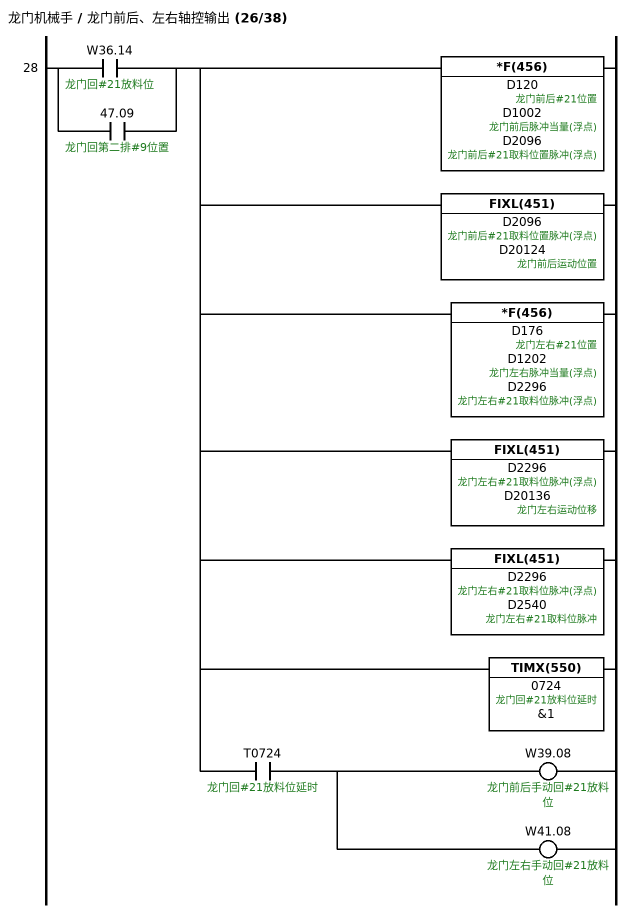
; [picture p353: 龙门机械手 / 龙门前后、左右轴控输出, rungs 28-28]
; rung 28
LD W36.14  ; 龙门回#21放料位
OR 47.09  ; 龙门回第二排#9位置
*F(456) D120 D1002 D2096  ; 龙门前后#21位置, 龙门前后脉冲当量(浮点), 龙门前后#21取料位置脉冲(浮点)
FIXL(451) D2096 D20124  ; 龙门前后#21取料位置脉冲(浮点), 龙门前后运动位置
*F(456) D176 D1202 D2296  ; 龙门左右#21位置, 龙门左右脉冲当量(浮点), 龙门左右#21取料位脉冲(浮点)
FIXL(451) D2296 D20136  ; 龙门左右#21取料位脉冲(浮点), 龙门左右运动位移
FIXL(451) D2296 D2540  ; 龙门左右#21取料位脉冲(浮点), 龙门左右#21取料位脉冲
TIMX(550) 0724 &1  ; 龙门回#21放料位延时
AND T0724  ; 龙门回#21放料位延时
OUT W39.08  ; 龙门前后手动回#21放料位
OUT W41.08  ; 龙门左右手动回#21放料位

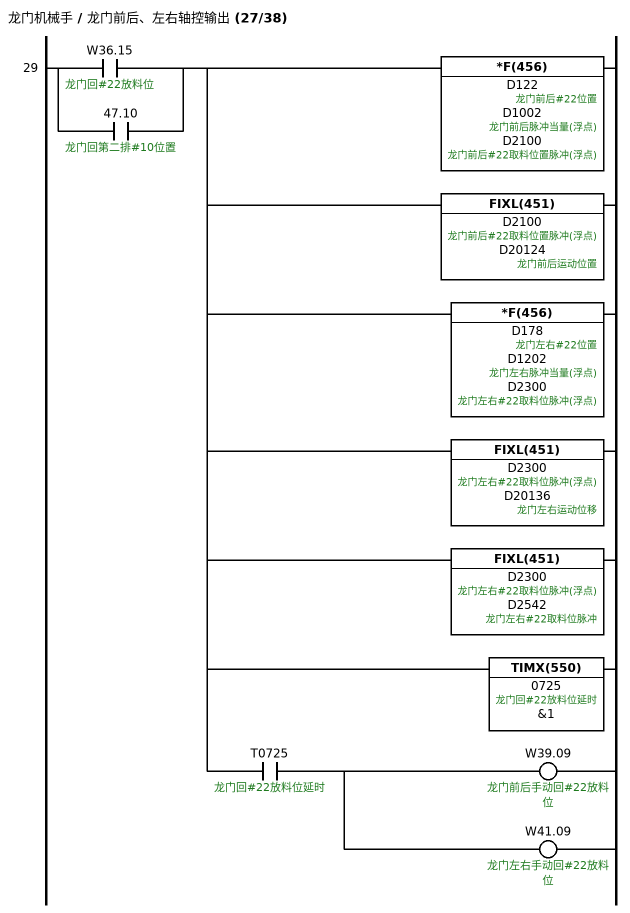
; rung 29
LD W36.15  ; 龙门回#22放料位
OR 47.10  ; 龙门回第二排#10位置
*F(456) D122 D1002 D2100  ; 龙门前后#22位置, 龙门前后脉冲当量(浮点), 龙门前后#22取料位置脉冲(浮点)
FIXL(451) D2100 D20124  ; 龙门前后#22取料位置脉冲(浮点), 龙门前后运动位置
*F(456) D178 D1202 D2300  ; 龙门左右#22位置, 龙门左右脉冲当量(浮点), 龙门左右#22取料位脉冲(浮点)
FIXL(451) D2300 D20136  ; 龙门左右#22取料位脉冲(浮点), 龙门左右运动位移
FIXL(451) D2300 D2542  ; 龙门左右#22取料位脉冲(浮点), 龙门左右#22取料位脉冲
TIMX(550) 0725 &1  ; 龙门回#22放料位延时
AND T0725  ; 龙门回#22放料位延时
OUT W39.09  ; 龙门前后手动回#22放料位
OUT W41.09  ; 龙门左右手动回#22放料位

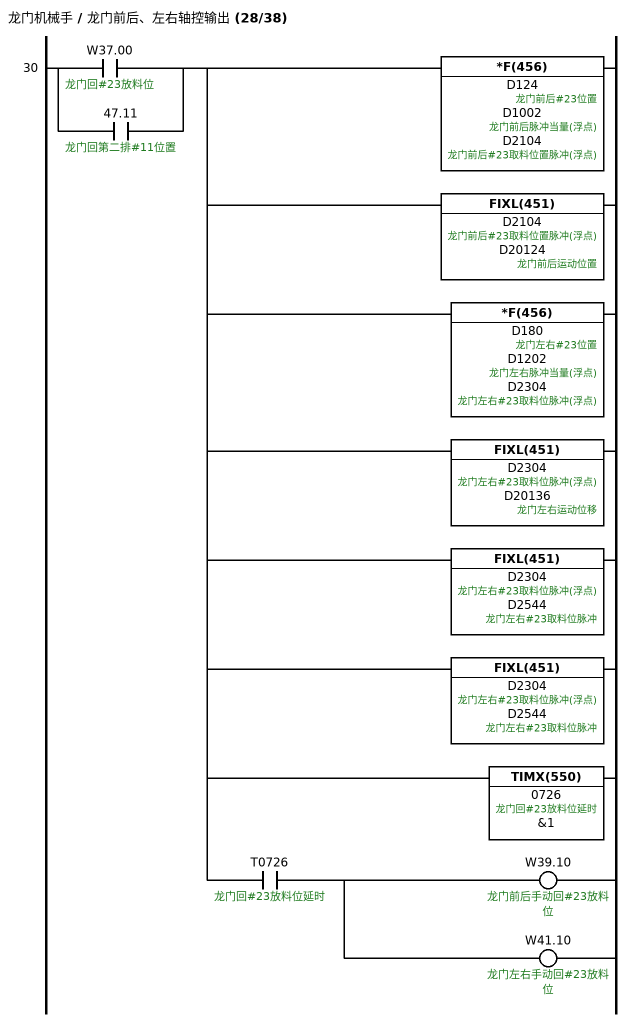
; rung 30
LD W37.00  ; 龙门回#23放料位
OR 47.11  ; 龙门回第二排#11位置
*F(456) D124 D1002 D2104  ; 龙门前后#23位置, 龙门前后脉冲当量(浮点), 龙门前后#23取料位置脉冲(浮点)
FIXL(451) D2104 D20124  ; 龙门前后#23取料位置脉冲(浮点), 龙门前后运动位置
*F(456) D180 D1202 D2304  ; 龙门左右#23位置, 龙门左右脉冲当量(浮点), 龙门左右#23取料位脉冲(浮点)
FIXL(451) D2304 D20136  ; 龙门左右#23取料位脉冲(浮点), 龙门左右运动位移
FIXL(451) D2304 D2544  ; 龙门左右#23取料位脉冲(浮点), 龙门左右#23取料位脉冲
FIXL(451) D2304 D2544  ; 龙门左右#23取料位脉冲(浮点), 龙门左右#23取料位脉冲
TIMX(550) 0726 &1  ; 龙门回#23放料位延时
AND T0726  ; 龙门回#23放料位延时
OUT W39.10  ; 龙门前后手动回#23放料位
OUT W41.10  ; 龙门左右手动回#23放料位

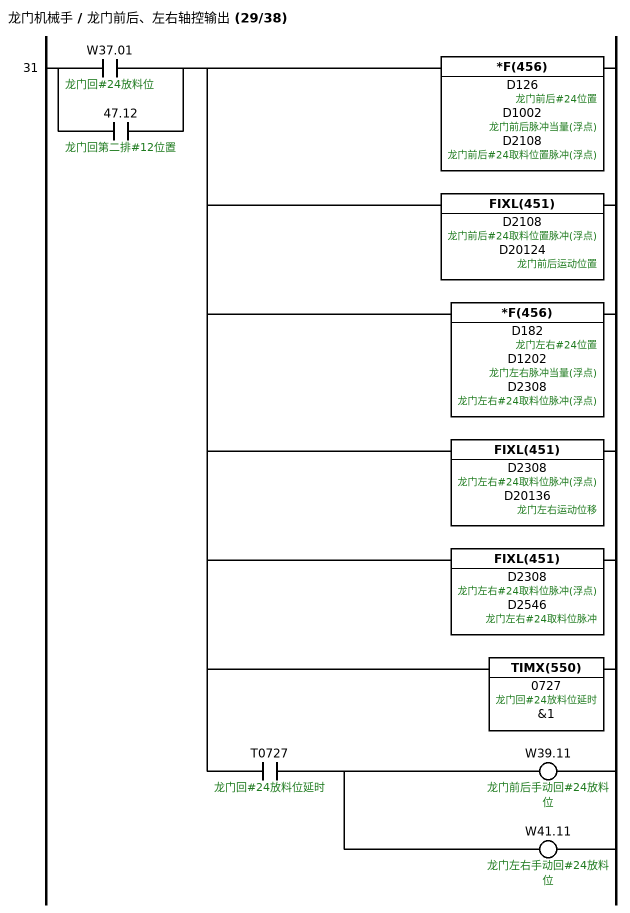
; rung 31
LD W37.01  ; 龙门回#24放料位
OR 47.12  ; 龙门回第二排#12位置
*F(456) D126 D1002 D2108  ; 龙门前后#24位置, 龙门前后脉冲当量(浮点), 龙门前后#24取料位置脉冲(浮点)
FIXL(451) D2108 D20124  ; 龙门前后#24取料位置脉冲(浮点), 龙门前后运动位置
*F(456) D182 D1202 D2308  ; 龙门左右#24位置, 龙门左右脉冲当量(浮点), 龙门左右#24取料位脉冲(浮点)
FIXL(451) D2308 D20136  ; 龙门左右#24取料位脉冲(浮点), 龙门左右运动位移
FIXL(451) D2308 D2546  ; 龙门左右#24取料位脉冲(浮点), 龙门左右#24取料位脉冲
TIMX(550) 0727 &1  ; 龙门回#24放料位延时
AND T0727  ; 龙门回#24放料位延时
OUT W39.11  ; 龙门前后手动回#24放料位
OUT W41.11  ; 龙门左右手动回#24放料位

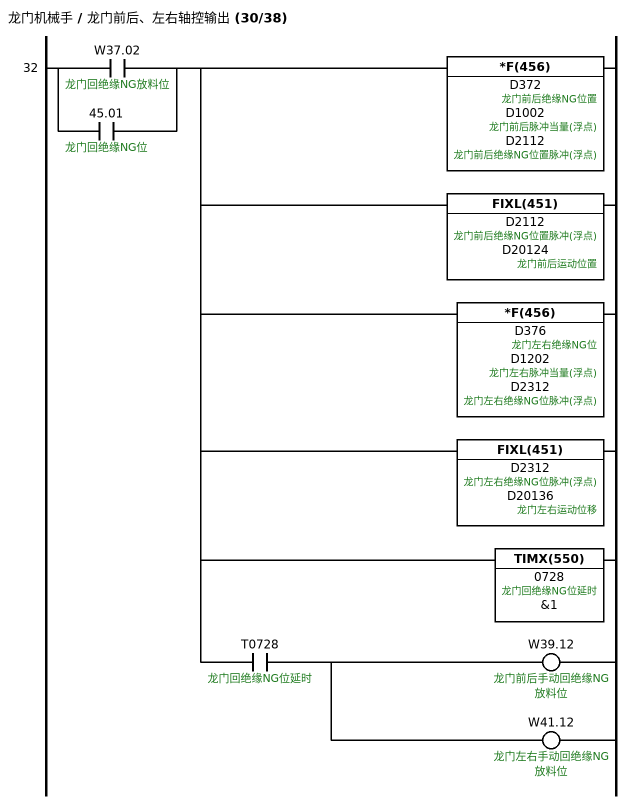
; rung 32
LD W37.02  ; 龙门回绝缘NG放料位
OR 45.01  ; 龙门回绝缘NG位
*F(456) D372 D1002 D2112  ; 龙门前后绝缘NG位置, 龙门前后脉冲当量(浮点), 龙门前后绝缘NG位置脉冲(浮点)
FIXL(451) D2112 D20124  ; 龙门前后绝缘NG位置脉冲(浮点), 龙门前后运动位置
*F(456) D376 D1202 D2312  ; 龙门左右绝缘NG位, 龙门左右脉冲当量(浮点), 龙门左右绝缘NG位脉冲(浮点)
FIXL(451) D2312 D20136  ; 龙门左右绝缘NG位脉冲(浮点), 龙门左右运动位移
TIMX(550) 0728 &1  ; 龙门回绝缘NG位延时
AND T0728  ; 龙门回绝缘NG位延时
OUT W39.12  ; 龙门前后手动回绝缘NG放料位
OUT W41.12  ; 龙门左右手动回绝缘NG放料位

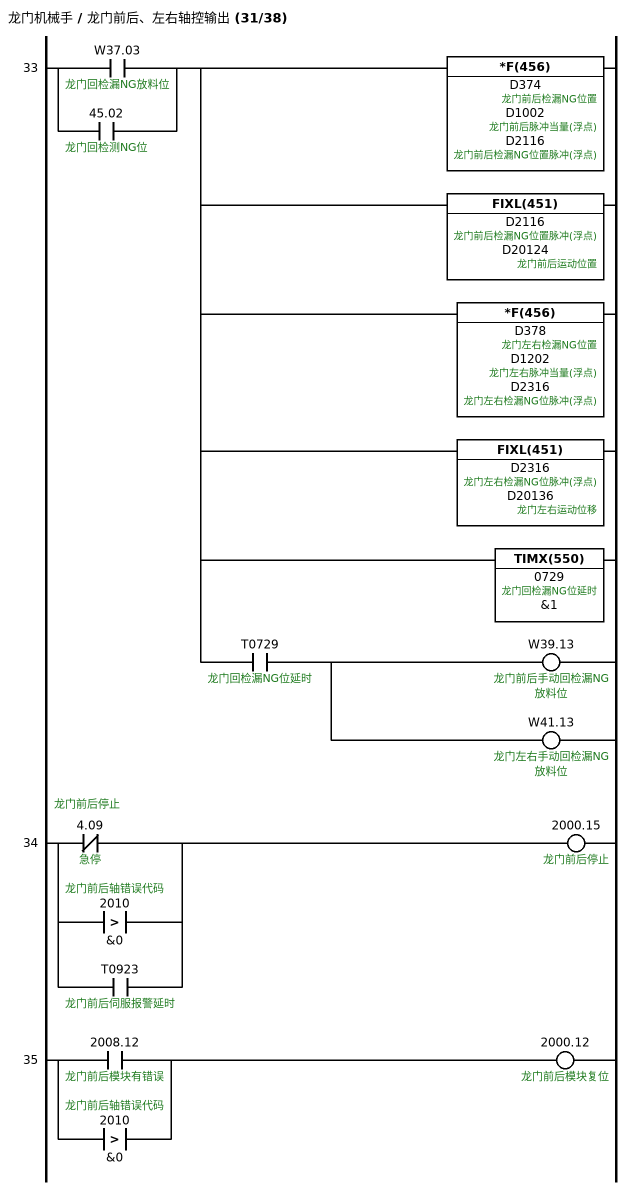
; rung 33
LD W37.03  ; 龙门回检漏NG放料位
OR 45.02  ; 龙门回检测NG位
*F(456) D374 D1002 D2116  ; 龙门前后检漏NG位置, 龙门前后脉冲当量(浮点), 龙门前后检漏NG位置脉冲(浮点)
FIXL(451) D2116 D20124  ; 龙门前后检漏NG位置脉冲(浮点), 龙门前后运动位置
*F(456) D378 D1202 D2316  ; 龙门左右检漏NG位置, 龙门左右脉冲当量(浮点), 龙门左右检漏NG位脉冲(浮点)
FIXL(451) D2316 D20136  ; 龙门左右检漏NG位脉冲(浮点), 龙门左右运动位移
TIMX(550) 0729 &1  ; 龙门回检漏NG位延时
AND T0729  ; 龙门回检漏NG位延时
OUT W39.13  ; 龙门前后手动回检漏NG放料位
OUT W41.13  ; 龙门左右手动回检漏NG放料位
; rung 34: 龙门前后停止
LDNOT 4.09  ; 急停
OR>(320) 2010 &0  ; 龙门前后轴错误代码
OR T0923  ; 龙门前后伺服报警延时
OUT 2000.15  ; 龙门前后停止
; rung 35
LD 2008.12  ; 龙门前后模块有错误
OR>(320) 2010 &0  ; 龙门前后轴错误代码
OUT 2000.12  ; 龙门前后模块复位

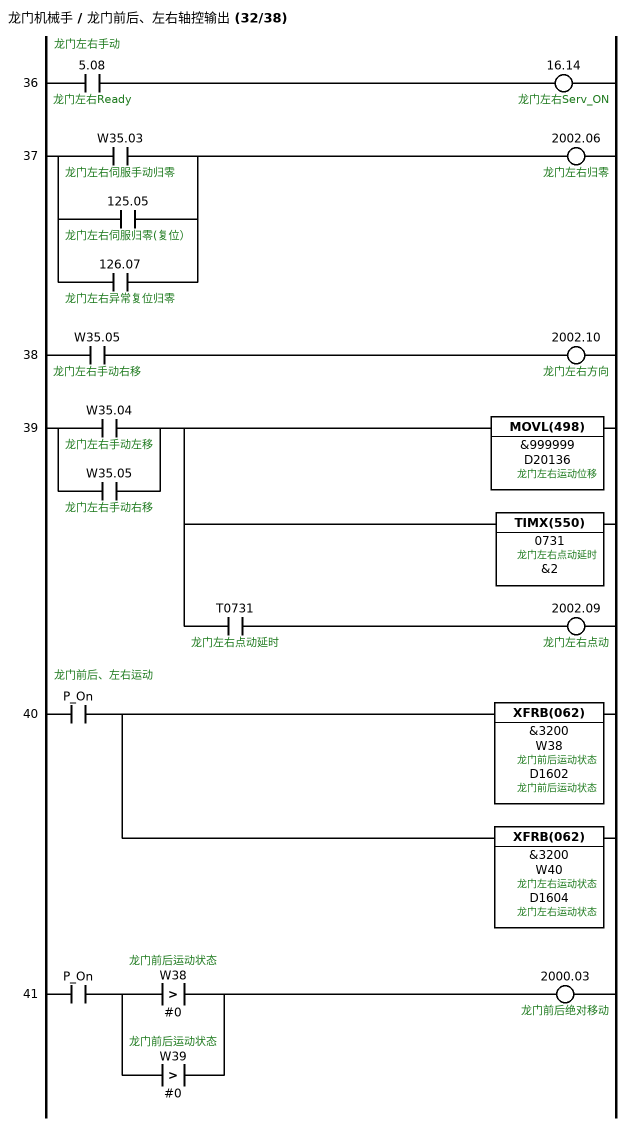
; rung 36: 龙门左右手动
LD 5.08  ; 龙门左右Ready
OUT 16.14  ; 龙门左右Serv_ON
; rung 37
LD W35.03  ; 龙门左右伺服手动归零
OR 125.05  ; 龙门左右伺服归零(复位）
OR 126.07  ; 龙门左右异常复位归零
OUT 2002.06  ; 龙门左右归零
; rung 38
LD W35.05  ; 龙门左右手动右移
OUT 2002.10  ; 龙门左右方向
; rung 39
LD W35.04  ; 龙门左右手动左移
OR W35.05  ; 龙门左右手动右移
MOVL(498) &999999 D20136  ; 龙门左右运动位移
TIMX(550) 0731 &2  ; 龙门左右点动延时
AND T0731  ; 龙门左右点动延时
OUT 2002.09  ; 龙门左右点动
; rung 40: 龙门前后、左右运动
LD P_On
XFRB(062) &3200 W38 D1602  ; 龙门前后运动状态
XFRB(062) &3200 W40 D1604  ; 龙门左右运动状态
; rung 41
LD P_On
LD>(320) W38 #0  ; 龙门前后运动状态
OR>(320) W39 #0  ; 龙门前后运动状态
ANDLD
OUT 2000.03  ; 龙门前后绝对移动

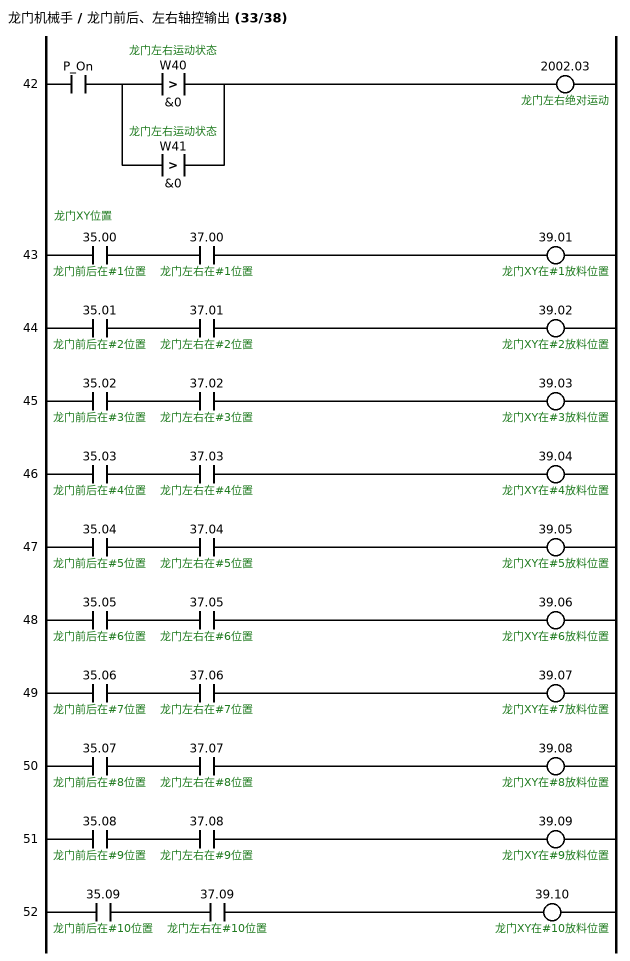
; rung 42
LD P_On
LD>(320) W40 &0  ; 龙门左右运动状态
OR>(320) W41 &0  ; 龙门左右运动状态
ANDLD
OUT 2002.03  ; 龙门左右绝对运动
; rung 43: 龙门XY位置
LD 35.00  ; 龙门前后在#1位置
AND 37.00  ; 龙门左右在#1位置
OUT 39.01  ; 龙门XY在#1放料位置
; rung 44
LD 35.01  ; 龙门前后在#2位置
AND 37.01  ; 龙门左右在#2位置
OUT 39.02  ; 龙门XY在#2放料位置
; rung 45
LD 35.02  ; 龙门前后在#3位置
AND 37.02  ; 龙门左右在#3位置
OUT 39.03  ; 龙门XY在#3放料位置
; rung 46
LD 35.03  ; 龙门前后在#4位置
AND 37.03  ; 龙门左右在#4位置
OUT 39.04  ; 龙门XY在#4放料位置
; rung 47
LD 35.04  ; 龙门前后在#5位置
AND 37.04  ; 龙门左右在#5位置
OUT 39.05  ; 龙门XY在#5放料位置
; rung 48
LD 35.05  ; 龙门前后在#6位置
AND 37.05  ; 龙门左右在#6位置
OUT 39.06  ; 龙门XY在#6放料位置
; rung 49
LD 35.06  ; 龙门前后在#7位置
AND 37.06  ; 龙门左右在#7位置
OUT 39.07  ; 龙门XY在#7放料位置
; rung 50
LD 35.07  ; 龙门前后在#8位置
AND 37.07  ; 龙门左右在#8位置
OUT 39.08  ; 龙门XY在#8放料位置
; rung 51
LD 35.08  ; 龙门前后在#9位置
AND 37.08  ; 龙门左右在#9位置
OUT 39.09  ; 龙门XY在#9放料位置
; rung 52
LD 35.09  ; 龙门前后在#10位置
AND 37.09  ; 龙门左右在#10位置
OUT 39.10  ; 龙门XY在#10放料位置

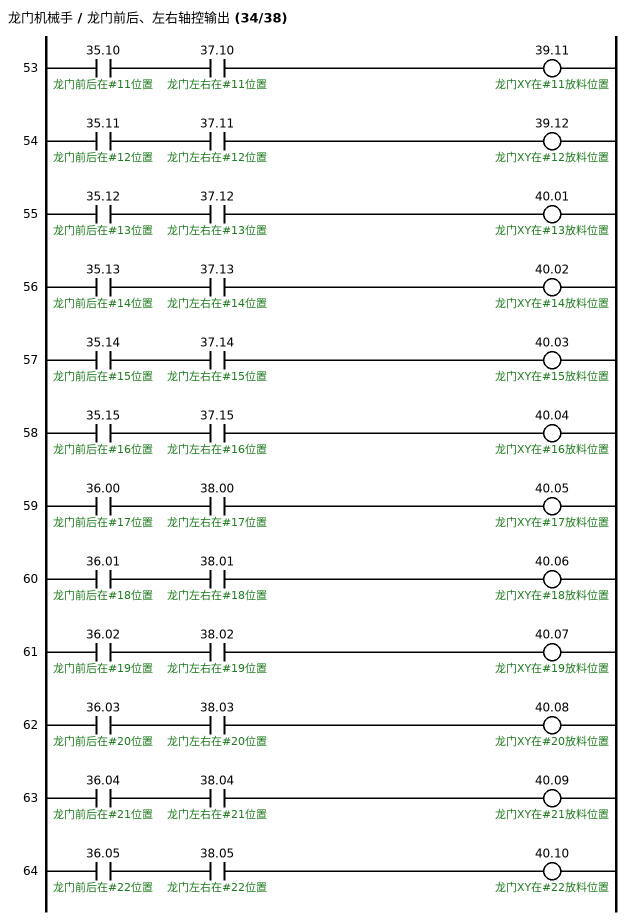
; rung 53
LD 35.10  ; 龙门前后在#11位置
AND 37.10  ; 龙门左右在#11位置
OUT 39.11  ; 龙门XY在#11放料位置
; rung 54
LD 35.11  ; 龙门前后在#12位置
AND 37.11  ; 龙门左右在#12位置
OUT 39.12  ; 龙门XY在#12放料位置
; rung 55
LD 35.12  ; 龙门前后在#13位置
AND 37.12  ; 龙门左右在#13位置
OUT 40.01  ; 龙门XY在#13放料位置
; rung 56
LD 35.13  ; 龙门前后在#14位置
AND 37.13  ; 龙门左右在#14位置
OUT 40.02  ; 龙门XY在#14放料位置
; rung 57
LD 35.14  ; 龙门前后在#15位置
AND 37.14  ; 龙门左右在#15位置
OUT 40.03  ; 龙门XY在#15放料位置
; rung 58
LD 35.15  ; 龙门前后在#16位置
AND 37.15  ; 龙门左右在#16位置
OUT 40.04  ; 龙门XY在#16放料位置
; rung 59
LD 36.00  ; 龙门前后在#17位置
AND 38.00  ; 龙门左右在#17位置
OUT 40.05  ; 龙门XY在#17放料位置
; rung 60
LD 36.01  ; 龙门前后在#18位置
AND 38.01  ; 龙门左右在#18位置
OUT 40.06  ; 龙门XY在#18放料位置
; rung 61
LD 36.02  ; 龙门前后在#19位置
AND 38.02  ; 龙门左右在#19位置
OUT 40.07  ; 龙门XY在#19放料位置
; rung 62
LD 36.03  ; 龙门前后在#20位置
AND 38.03  ; 龙门左右在#20位置
OUT 40.08  ; 龙门XY在#20放料位置
; rung 63
LD 36.04  ; 龙门前后在#21位置
AND 38.04  ; 龙门左右在#21位置
OUT 40.09  ; 龙门XY在#21放料位置
; rung 64
LD 36.05  ; 龙门前后在#22位置
AND 38.05  ; 龙门左右在#22位置
OUT 40.10  ; 龙门XY在#22放料位置

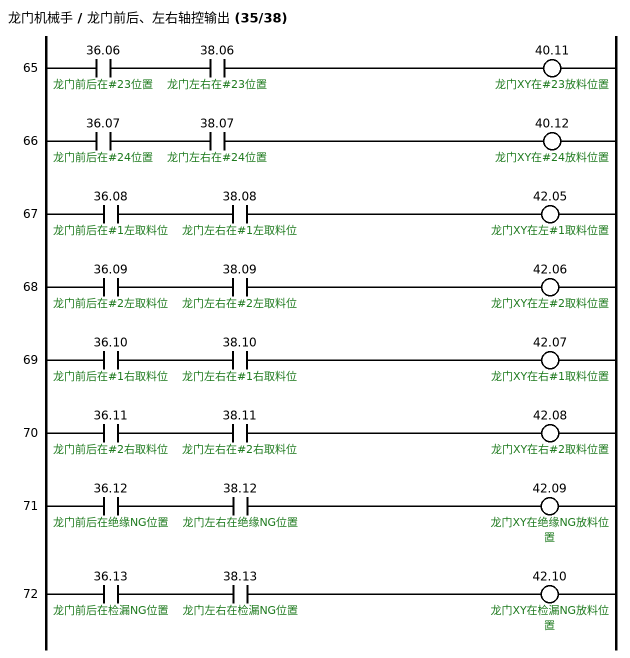
; rung 65
LD 36.06  ; 龙门前后在#23位置
AND 38.06  ; 龙门左右在#23位置
OUT 40.11  ; 龙门XY在#23放料位置
; rung 66
LD 36.07  ; 龙门前后在#24位置
AND 38.07  ; 龙门左右在#24位置
OUT 40.12  ; 龙门XY在#24放料位置
; rung 67
LD 36.08  ; 龙门前后在#1左取料位
AND 38.08  ; 龙门左右在#1左取料位
OUT 42.05  ; 龙门XY在左#1取料位置
; rung 68
LD 36.09  ; 龙门前后在#2左取料位
AND 38.09  ; 龙门左右在#2左取料位
OUT 42.06  ; 龙门XY在左#2取料位置
; rung 69
LD 36.10  ; 龙门前后在#1右取料位
AND 38.10  ; 龙门左右在#1右取料位
OUT 42.07  ; 龙门XY在右#1取料位置
; rung 70
LD 36.11  ; 龙门前后在#2右取料位
AND 38.11  ; 龙门左右在#2右取料位
OUT 42.08  ; 龙门XY在右#2取料位置
; rung 71
LD 36.12  ; 龙门前后在绝缘NG位置
AND 38.12  ; 龙门左右在绝缘NG位置
OUT 42.09  ; 龙门XY在绝缘NG放料位置
; rung 72
LD 36.13  ; 龙门前后在检漏NG位置
AND 38.13  ; 龙门左右在检漏NG位置
OUT 42.10  ; 龙门XY在检漏NG放料位置

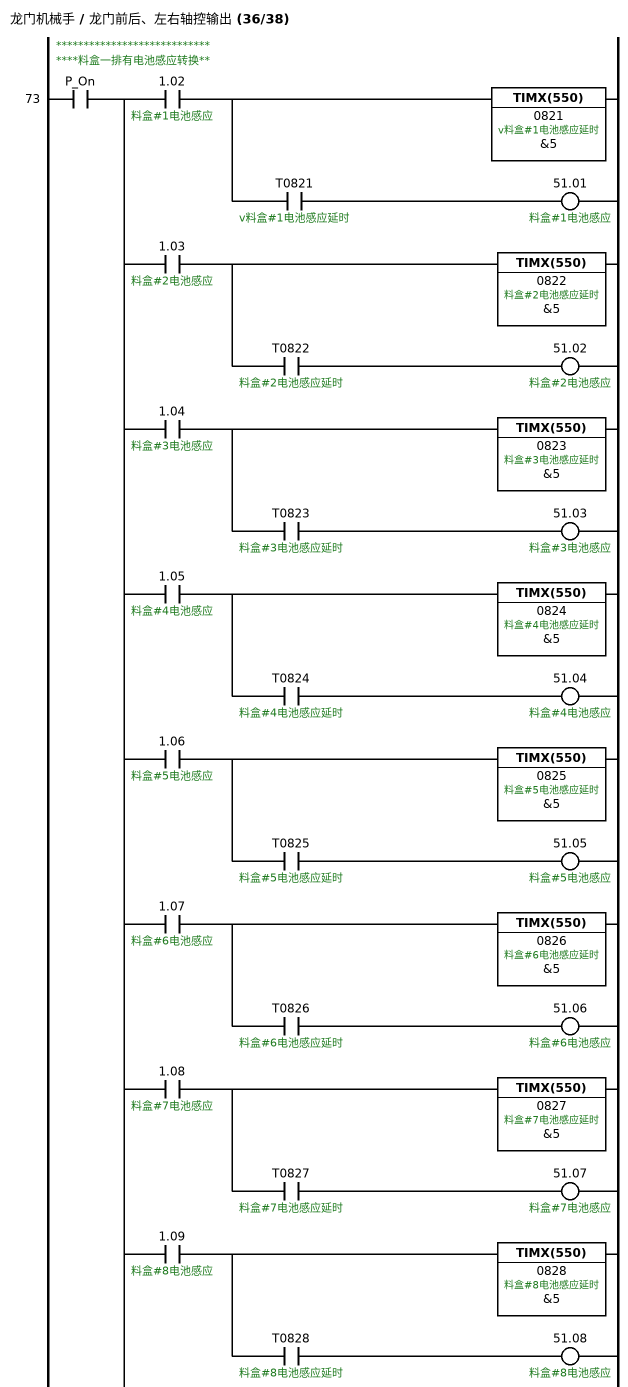

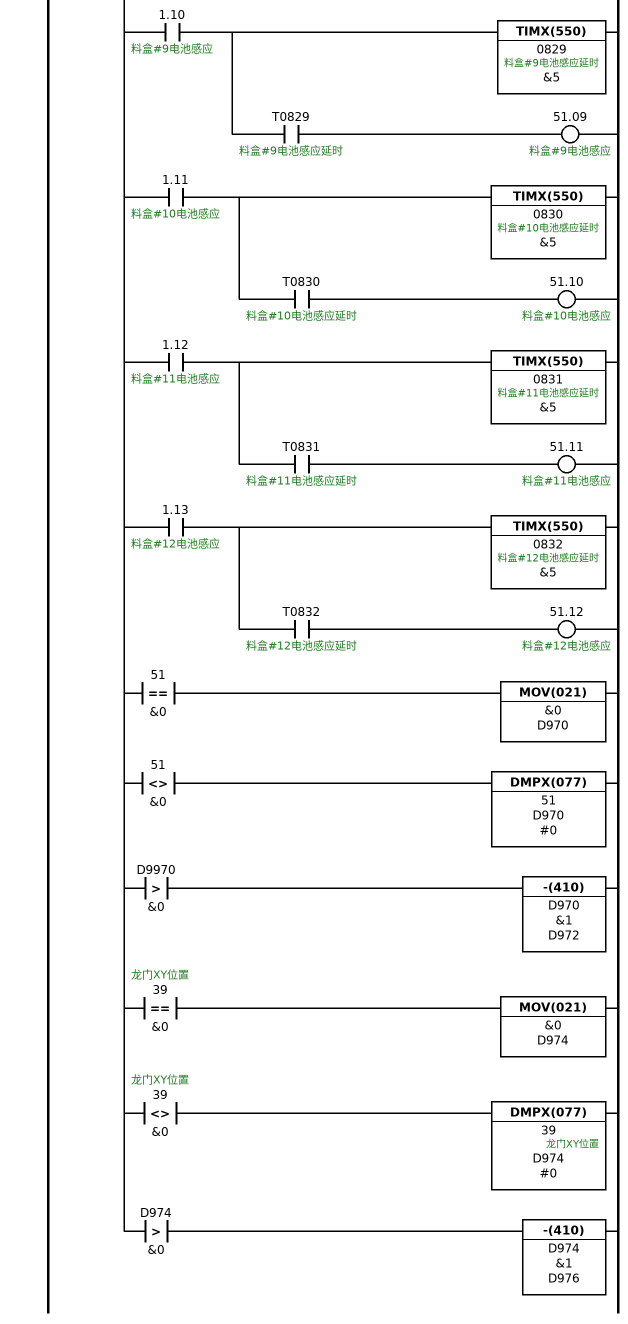
; rung 73: **************************** / ****料盒一排有电池感应转换**
LD P_On
OUT TR0
AND 1.02  ; 料盒#1电池感应
TIMX(550) 0821 &5  ; v料盒#1电池感应延时
AND T0821  ; v料盒#1电池感应延时
OUT 51.01  ; 料盒#1电池感应
LD TR0
AND 1.03  ; 料盒#2电池感应
TIMX(550) 0822 &5  ; 料盒#2电池感应延时
AND T0822  ; 料盒#2电池感应延时
OUT 51.02  ; 料盒#2电池感应
LD TR0
AND 1.04  ; 料盒#3电池感应
TIMX(550) 0823 &5  ; 料盒#3电池感应延时
AND T0823  ; 料盒#3电池感应延时
OUT 51.03  ; 料盒#3电池感应
LD TR0
AND 1.05  ; 料盒#4电池感应
TIMX(550) 0824 &5  ; 料盒#4电池感应延时
AND T0824  ; 料盒#4电池感应延时
OUT 51.04  ; 料盒#4电池感应
LD TR0
AND 1.06  ; 料盒#5电池感应
TIMX(550) 0825 &5  ; 料盒#5电池感应延时
AND T0825  ; 料盒#5电池感应延时
OUT 51.05  ; 料盒#5电池感应
LD TR0
AND 1.07  ; 料盒#6电池感应
TIMX(550) 0826 &5  ; 料盒#6电池感应延时
AND T0826  ; 料盒#6电池感应延时
OUT 51.06  ; 料盒#6电池感应
LD TR0
AND 1.08  ; 料盒#7电池感应
TIMX(550) 0827 &5  ; 料盒#7电池感应延时
AND T0827  ; 料盒#7电池感应延时
OUT 51.07  ; 料盒#7电池感应
LD TR0
AND 1.09  ; 料盒#8电池感应
TIMX(550) 0828 &5  ; 料盒#8电池感应延时
AND T0828  ; 料盒#8电池感应延时
OUT 51.08  ; 料盒#8电池感应
LD TR0
AND 1.10  ; 料盒#9电池感应
TIMX(550) 0829 &5  ; 料盒#9电池感应延时
AND T0829  ; 料盒#9电池感应延时
OUT 51.09  ; 料盒#9电池感应
LD TR0
AND 1.11  ; 料盒#10电池感应
TIMX(550) 0830 &5  ; 料盒#10电池感应延时
AND T0830  ; 料盒#10电池感应延时
OUT 51.10  ; 料盒#10电池感应
LD TR0
AND 1.12  ; 料盒#11电池感应
TIMX(550) 0831 &5  ; 料盒#11电池感应延时
AND T0831  ; 料盒#11电池感应延时
OUT 51.11  ; 料盒#11电池感应
LD TR0
AND 1.13  ; 料盒#12电池感应
TIMX(550) 0832 &5  ; 料盒#12电池感应延时
AND T0832  ; 料盒#12电池感应延时
OUT 51.12  ; 料盒#12电池感应
LD TR0
AND=(300) 51 &0
MOV(021) &0 D970
LD TR0
AND<>(305) 51 &0
DMPX(077) 51 D970 #0
LD TR0
AND>(320) D9970 &0
-(410) D970 &1 D972
LD TR0
AND=(300) 39 &0  ; 龙门XY位置
MOV(021) &0 D974
LD TR0
AND<>(305) 39 &0  ; 龙门XY位置
DMPX(077) 39 D974 #0  ; 龙门XY位置
LD TR0
AND>(320) D974 &0
-(410) D974 &1 D976

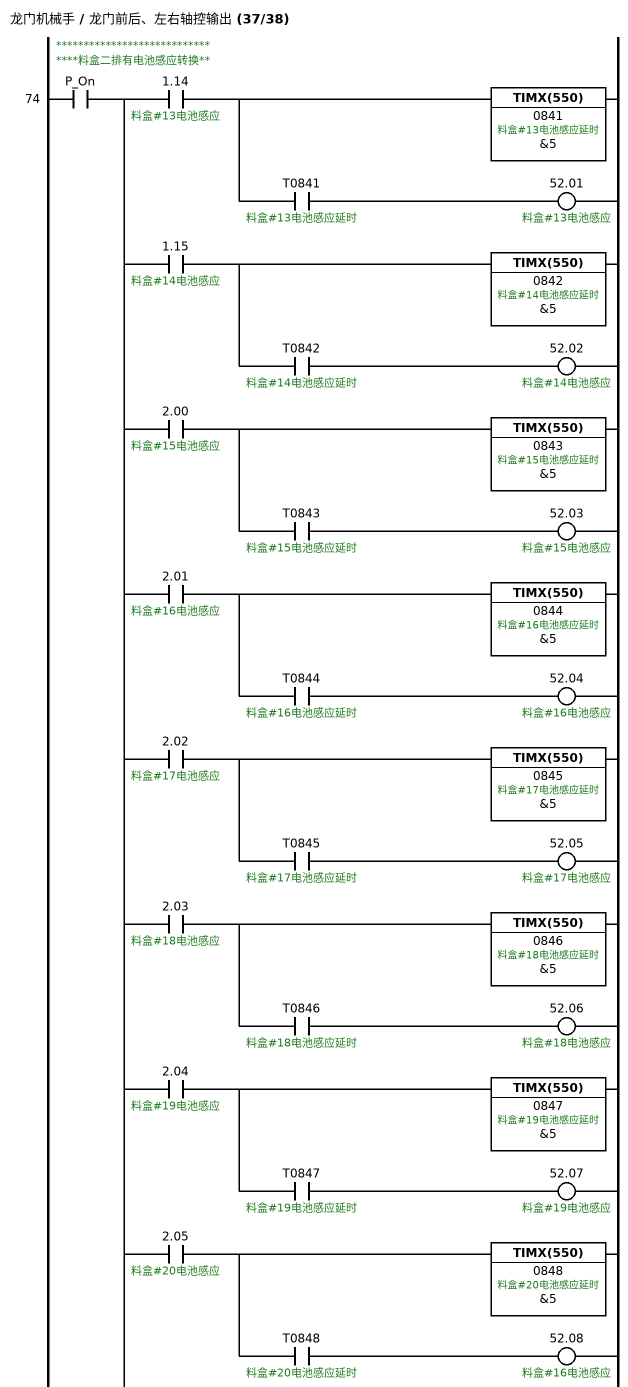

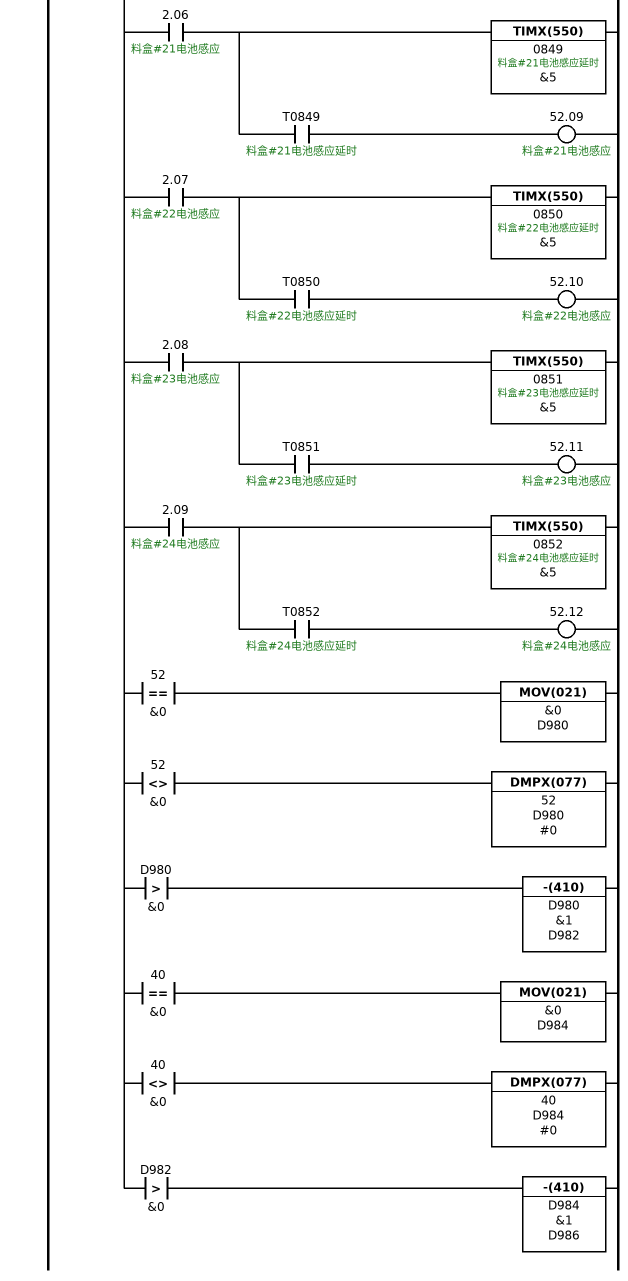
; rung 74: **************************** / ****料盒二排有电池感应转换**
LD P_On
OUT TR0
AND 1.14  ; 料盒#13电池感应
TIMX(550) 0841 &5  ; 料盒#13电池感应延时
AND T0841  ; 料盒#13电池感应延时
OUT 52.01  ; 料盒#13电池感应
LD TR0
AND 1.15  ; 料盒#14电池感应
TIMX(550) 0842 &5  ; 料盒#14电池感应延时
AND T0842  ; 料盒#14电池感应延时
OUT 52.02  ; 料盒#14电池感应
LD TR0
AND 2.00  ; 料盒#15电池感应
TIMX(550) 0843 &5  ; 料盒#15电池感应延时
AND T0843  ; 料盒#15电池感应延时
OUT 52.03  ; 料盒#15电池感应
LD TR0
AND 2.01  ; 料盒#16电池感应
TIMX(550) 0844 &5  ; 料盒#16电池感应延时
AND T0844  ; 料盒#16电池感应延时
OUT 52.04  ; 料盒#16电池感应
LD TR0
AND 2.02  ; 料盒#17电池感应
TIMX(550) 0845 &5  ; 料盒#17电池感应延时
AND T0845  ; 料盒#17电池感应延时
OUT 52.05  ; 料盒#17电池感应
LD TR0
AND 2.03  ; 料盒#18电池感应
TIMX(550) 0846 &5  ; 料盒#18电池感应延时
AND T0846  ; 料盒#18电池感应延时
OUT 52.06  ; 料盒#18电池感应
LD TR0
AND 2.04  ; 料盒#19电池感应
TIMX(550) 0847 &5  ; 料盒#19电池感应延时
AND T0847  ; 料盒#19电池感应延时
OUT 52.07  ; 料盒#19电池感应
LD TR0
AND 2.05  ; 料盒#20电池感应
TIMX(550) 0848 &5  ; 料盒#20电池感应延时
AND T0848  ; 料盒#20电池感应延时
OUT 52.08  ; 料盒#16电池感应
LD TR0
AND 2.06  ; 料盒#21电池感应
TIMX(550) 0849 &5  ; 料盒#21电池感应延时
AND T0849  ; 料盒#21电池感应延时
OUT 52.09  ; 料盒#21电池感应
LD TR0
AND 2.07  ; 料盒#22电池感应
TIMX(550) 0850 &5  ; 料盒#22电池感应延时
AND T0850  ; 料盒#22电池感应延时
OUT 52.10  ; 料盒#22电池感应
LD TR0
AND 2.08  ; 料盒#23电池感应
TIMX(550) 0851 &5  ; 料盒#23电池感应延时
AND T0851  ; 料盒#23电池感应延时
OUT 52.11  ; 料盒#23电池感应
LD TR0
AND 2.09  ; 料盒#24电池感应
TIMX(550) 0852 &5  ; 料盒#24电池感应延时
AND T0852  ; 料盒#24电池感应延时
OUT 52.12  ; 料盒#24电池感应
LD TR0
AND=(300) 52 &0
MOV(021) &0 D980
LD TR0
AND<>(305) 52 &0
DMPX(077) 52 D980 #0
LD TR0
AND>(320) D980 &0
-(410) D980 &1 D982
LD TR0
AND=(300) 40 &0
MOV(021) &0 D984
LD TR0
AND<>(305) 40 &0
DMPX(077) 40 D984 #0
LD TR0
AND>(320) D982 &0
-(410) D984 &1 D986

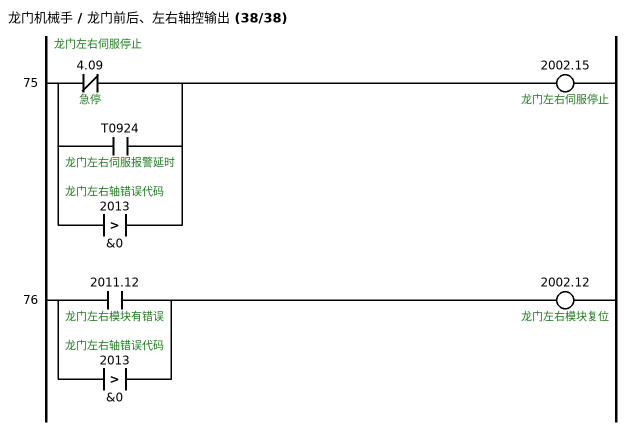
; rung 75: 龙门左右伺服停止
LDNOT 4.09  ; 急停
OR T0924  ; 龙门左右伺服报警延时
OR>(320) 2013 &0  ; 龙门左右轴错误代码
OUT 2002.15  ; 龙门左右伺服停止
; rung 76
LD 2011.12  ; 龙门左右模块有错误
OR>(320) 2013 &0  ; 龙门左右轴错误代码
OUT 2002.12  ; 龙门左右模块复位

### Section 龙门、料盒升降轴控输出

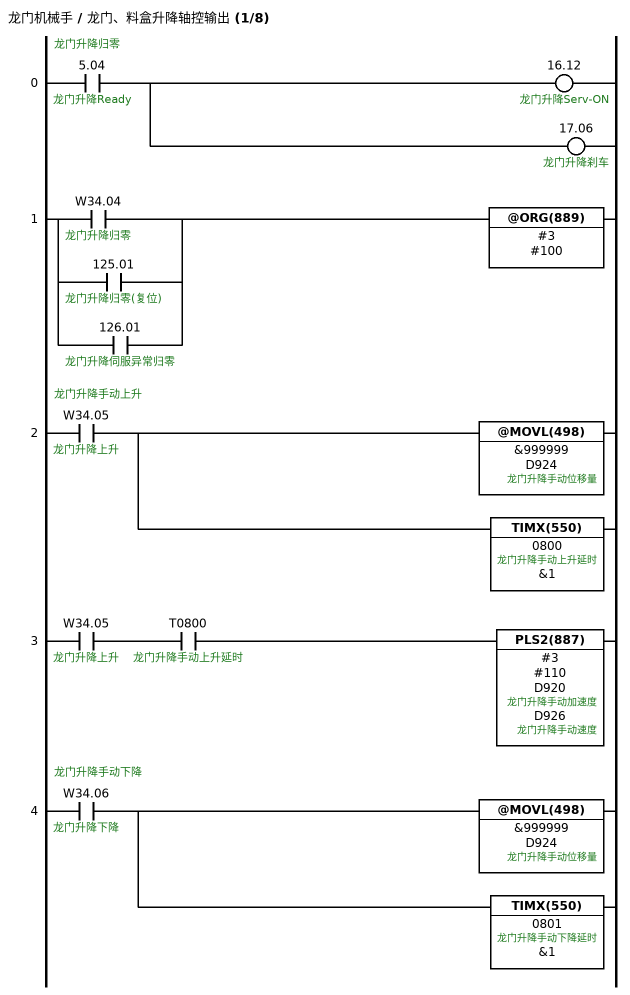
; rung 0: 龙门升降归零
LD 5.04  ; 龙门升降Ready
OUT 16.12  ; 龙门升降Serv-ON
OUT 17.06  ; 龙门升降刹车
; rung 1
LD W34.04  ; 龙门升降归零
OR 125.01  ; 龙门升降归零(复位)
OR 126.01  ; 龙门升降伺服异常归零
@ORG(889) #3 #100
; rung 2: 龙门升降手动上升
LD W34.05  ; 龙门升降上升
@MOVL(498) &999999 D924  ; 龙门升降手动位移量
TIMX(550) 0800 &1  ; 龙门升降手动上升延时
; rung 3
LD W34.05  ; 龙门升降上升
AND T0800  ; 龙门升降手动上升延时
PLS2(887) #3 #110 D920 D926  ; 龙门升降手动加速度, 龙门升降手动速度
; rung 4: 龙门升降手动下降
LD W34.06  ; 龙门升降下降
@MOVL(498) &999999 D924  ; 龙门升降手动位移量
TIMX(550) 0801 &1  ; 龙门升降手动下降延时

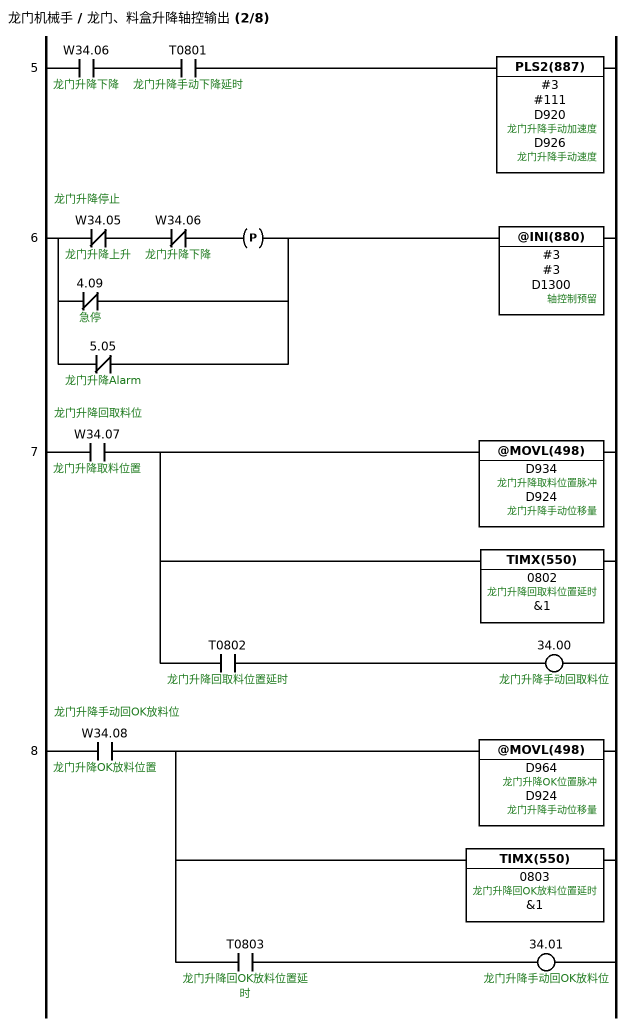
; rung 5
LD W34.06  ; 龙门升降下降
AND T0801  ; 龙门升降手动下降延时
PLS2(887) #3 #111 D920 D926  ; 龙门升降手动加速度, 龙门升降手动速度
; rung 6: 龙门升降停止
LDNOT W34.05  ; 龙门升降上升
ANDNOT W34.06  ; 龙门升降下降
UP(521)
ORNOT 4.09  ; 急停
ORNOT 5.05  ; 龙门升降Alarm
@INI(880) #3 #3 D1300  ; 轴控制预留
; rung 7: 龙门升降回取料位
LD W34.07  ; 龙门升降取料位置
@MOVL(498) D934 D924  ; 龙门升降取料位置脉冲, 龙门升降手动位移量
TIMX(550) 0802 &1  ; 龙门升降回取料位置延时
AND T0802  ; 龙门升降回取料位置延时
OUT 34.00  ; 龙门升降手动回取料位
; rung 8: 龙门升降手动回OK放料位
LD W34.08  ; 龙门升降OK放料位置
@MOVL(498) D964 D924  ; 龙门升降OK位置脉冲, 龙门升降手动位移量
TIMX(550) 0803 &1  ; 龙门升降回OK放料位置延时
AND T0803  ; 龙门升降回OK放料位置延时
OUT 34.01  ; 龙门升降手动回OK放料位

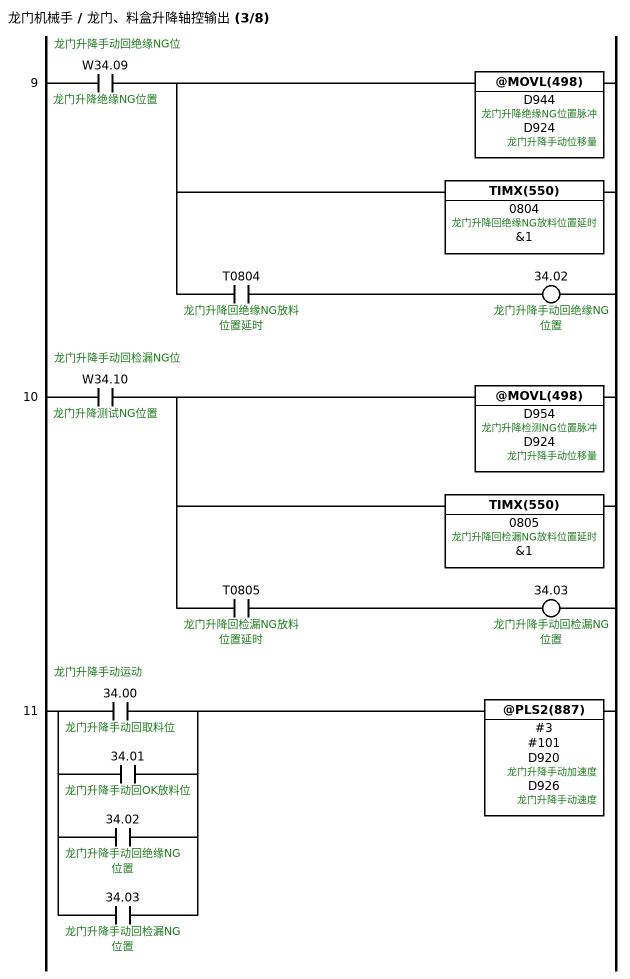
; rung 9: 龙门升降手动回绝缘NG位
LD W34.09  ; 龙门升降绝缘NG位置
@MOVL(498) D944 D924  ; 龙门升降绝缘NG位置脉冲, 龙门升降手动位移量
TIMX(550) 0804 &1  ; 龙门升降回绝缘NG放料位置延时
AND T0804  ; 龙门升降回绝缘NG放料位置延时
OUT 34.02  ; 龙门升降手动回绝缘NG位置
; rung 10: 龙门升降手动回检漏NG位
LD W34.10  ; 龙门升降测试NG位置
@MOVL(498) D954 D924  ; 龙门升降检测NG位置脉冲, 龙门升降手动位移量
TIMX(550) 0805 &1  ; 龙门升降回检漏NG放料位置延时
AND T0805  ; 龙门升降回检漏NG放料位置延时
OUT 34.03  ; 龙门升降手动回检漏NG位置
; rung 11: 龙门升降手动运动
LD 34.00  ; 龙门升降手动回取料位
OR 34.01  ; 龙门升降手动回OK放料位
OR 34.02  ; 龙门升降手动回绝缘NG位置
OR 34.03  ; 龙门升降手动回检漏NG位置
@PLS2(887) #3 #101 D920 D926  ; 龙门升降手动加速度, 龙门升降手动速度

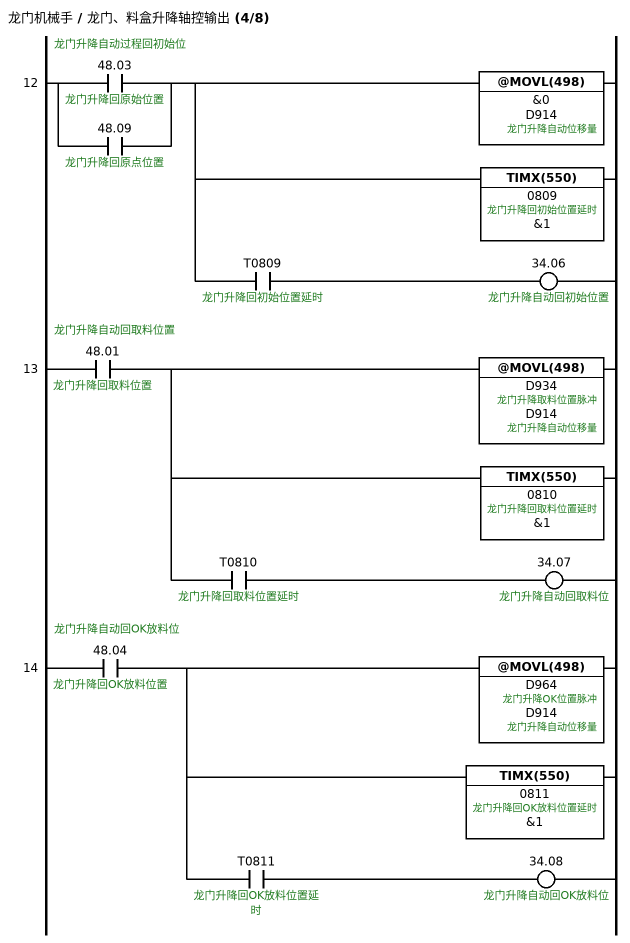
; rung 12: 龙门升降自动过程回初始位
LD 48.03  ; 龙门升降回原始位置
OR 48.09  ; 龙门升降回原点位置
@MOVL(498) &0 D914  ; 龙门升降自动位移量
TIMX(550) 0809 &1  ; 龙门升降回初始位置延时
AND T0809  ; 龙门升降回初始位置延时
OUT 34.06  ; 龙门升降自动回初始位置
; rung 13: 龙门升降自动回取料位置
LD 48.01  ; 龙门升降回取料位置
@MOVL(498) D934 D914  ; 龙门升降取料位置脉冲, 龙门升降自动位移量
TIMX(550) 0810 &1  ; 龙门升降回取料位置延时
AND T0810  ; 龙门升降回取料位置延时
OUT 34.07  ; 龙门升降自动回取料位
; rung 14: 龙门升降自动回OK放料位
LD 48.04  ; 龙门升降回OK放料位置
@MOVL(498) D964 D914  ; 龙门升降OK位置脉冲, 龙门升降自动位移量
TIMX(550) 0811 &1  ; 龙门升降回OK放料位置延时
AND T0811  ; 龙门升降回OK放料位置延时
OUT 34.08  ; 龙门升降自动回OK放料位

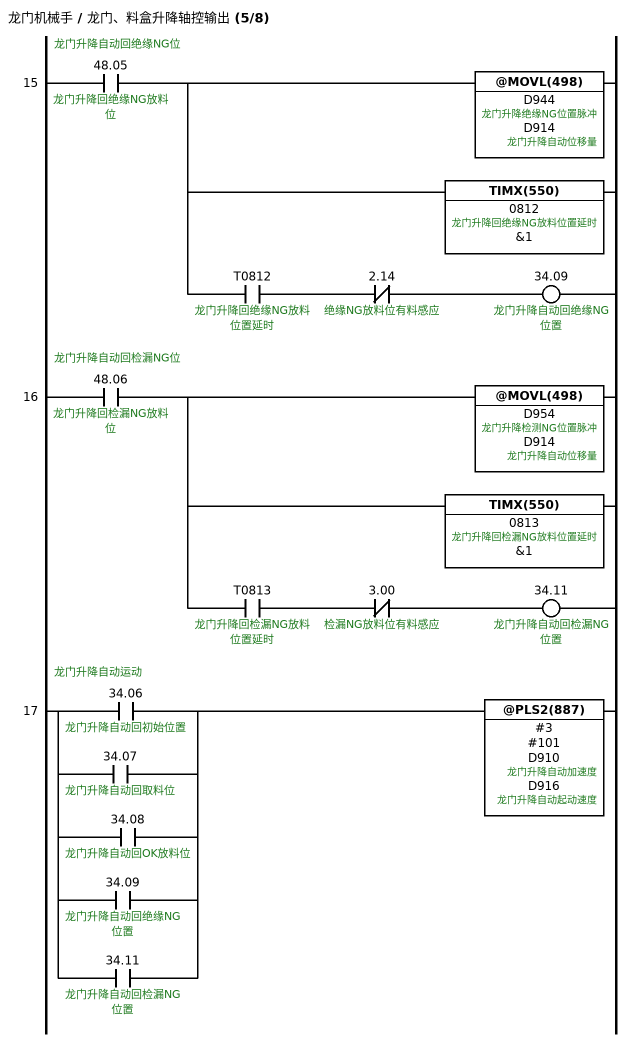
; rung 15: 龙门升降自动回绝缘NG位
LD 48.05  ; 龙门升降回绝缘NG放料位
@MOVL(498) D944 D914  ; 龙门升降绝缘NG位置脉冲, 龙门升降自动位移量
TIMX(550) 0812 &1  ; 龙门升降回绝缘NG放料位置延时
AND T0812  ; 龙门升降回绝缘NG放料位置延时
ANDNOT 2.14  ; 绝缘NG放料位有料感应
OUT 34.09  ; 龙门升降自动回绝缘NG位置
; rung 16: 龙门升降自动回检漏NG位
LD 48.06  ; 龙门升降回检漏NG放料位
@MOVL(498) D954 D914  ; 龙门升降检测NG位置脉冲, 龙门升降自动位移量
TIMX(550) 0813 &1  ; 龙门升降回检漏NG放料位置延时
AND T0813  ; 龙门升降回检漏NG放料位置延时
ANDNOT 3.00  ; 检漏NG放料位有料感应
OUT 34.11  ; 龙门升降自动回检漏NG位置
; rung 17: 龙门升降自动运动
LD 34.06  ; 龙门升降自动回初始位置
OR 34.07  ; 龙门升降自动回取料位
OR 34.08  ; 龙门升降自动回OK放料位
OR 34.09  ; 龙门升降自动回绝缘NG位置
OR 34.11  ; 龙门升降自动回检漏NG位置
@PLS2(887) #3 #101 D910 D916  ; 龙门升降自动加速度, 龙门升降自动起动速度

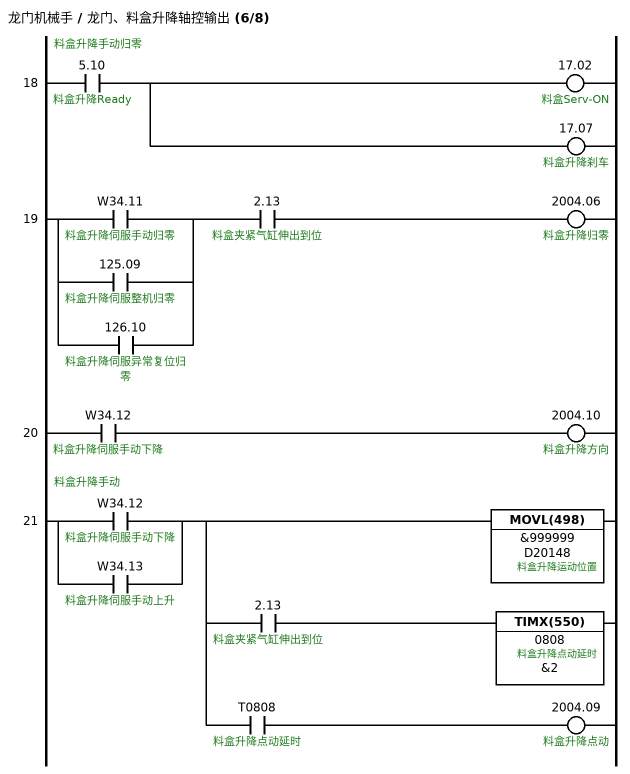
; rung 18: 料盒升降手动归零
LD 5.10  ; 料盒升降Ready
OUT 17.02  ; 料盒Serv-ON
OUT 17.07  ; 料盒升降刹车
; rung 19
LD W34.11  ; 料盒升降伺服手动归零
OR 125.09  ; 料盒升降伺服整机归零
OR 126.10  ; 料盒升降伺服异常复位归零
AND 2.13  ; 料盒夹紧气缸伸出到位
OUT 2004.06  ; 料盒升降归零
; rung 20
LD W34.12  ; 料盒升降伺服手动下降
OUT 2004.10  ; 料盒升降方向
; rung 21: 料盒升降手动
LD W34.12  ; 料盒升降伺服手动下降
OR W34.13  ; 料盒升降伺服手动上升
OUT TR0
MOVL(498) &999999 D20148  ; 料盒升降运动位置
AND 2.13  ; 料盒夹紧气缸伸出到位
TIMX(550) 0808 &2  ; 料盒升降点动延时
LD TR0
AND T0808  ; 料盒升降点动延时
OUT 2004.09  ; 料盒升降点动

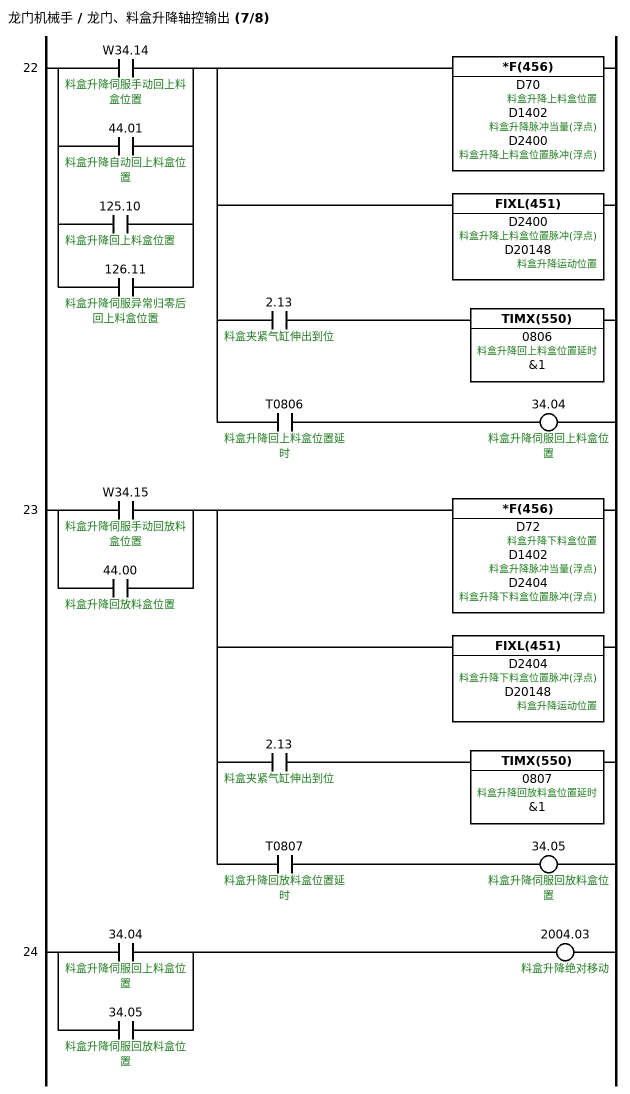
; rung 22
LD W34.14  ; 料盒升降伺服手动回上料盒位置
OR 44.01  ; 料盒升降自动回上料盒位置
OR 125.10  ; 料盒升降回上料盒位置
OR 126.11  ; 料盒升降伺服异常归零后回上料盒位置
OUT TR0
*F(456) D70 D1402 D2400  ; 料盒升降上料盒位置, 料盒升降脉冲当量(浮点), 料盒升降上料盒位置脉冲(浮点)
FIXL(451) D2400 D20148  ; 料盒升降上料盒位置脉冲(浮点), 料盒升降运动位置
AND 2.13  ; 料盒夹紧气缸伸出到位
TIMX(550) 0806 &1  ; 料盒升降回上料盒位置延时
LD TR0
AND T0806  ; 料盒升降回上料盒位置延时
OUT 34.04  ; 料盒升降伺服回上料盒位置
; rung 23
LD W34.15  ; 料盒升降伺服手动回放料盒位置
OR 44.00  ; 料盒升降回放料盒位置
OUT TR0
*F(456) D72 D1402 D2404  ; 料盒升降下料盒位置, 料盒升降脉冲当量(浮点), 料盒升降下料盒位置脉冲(浮点)
FIXL(451) D2404 D20148  ; 料盒升降下料盒位置脉冲(浮点), 料盒升降运动位置
AND 2.13  ; 料盒夹紧气缸伸出到位
TIMX(550) 0807 &1  ; 料盒升降回放料盒位置延时
LD TR0
AND T0807  ; 料盒升降回放料盒位置延时
OUT 34.05  ; 料盒升降伺服回放料盒位置
; rung 24
LD 34.04  ; 料盒升降伺服回上料盒位置
OR 34.05  ; 料盒升降伺服回放料盒位置
OUT 2004.03  ; 料盒升降绝对移动

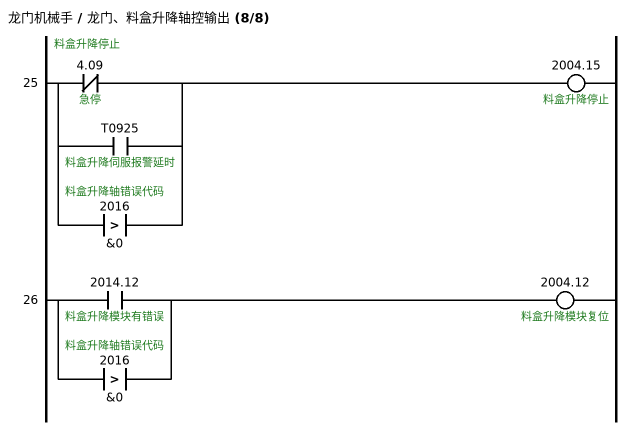
; rung 25: 料盒升降停止
LDNOT 4.09  ; 急停
OR T0925  ; 料盒升降伺服报警延时
OR>(320) 2016 &0  ; 料盒升降轴错误代码
OUT 2004.15  ; 料盒升降停止
; rung 26
LD 2014.12  ; 料盒升降模块有错误
OR>(320) 2016 &0  ; 料盒升降轴错误代码
OUT 2004.12  ; 料盒升降模块复位

### Section END
; rung 0
END(001)

## Program 龙门机构 (cyclic task 8)
Local symbols
f114 BOOL

### Section 龙门机构手动

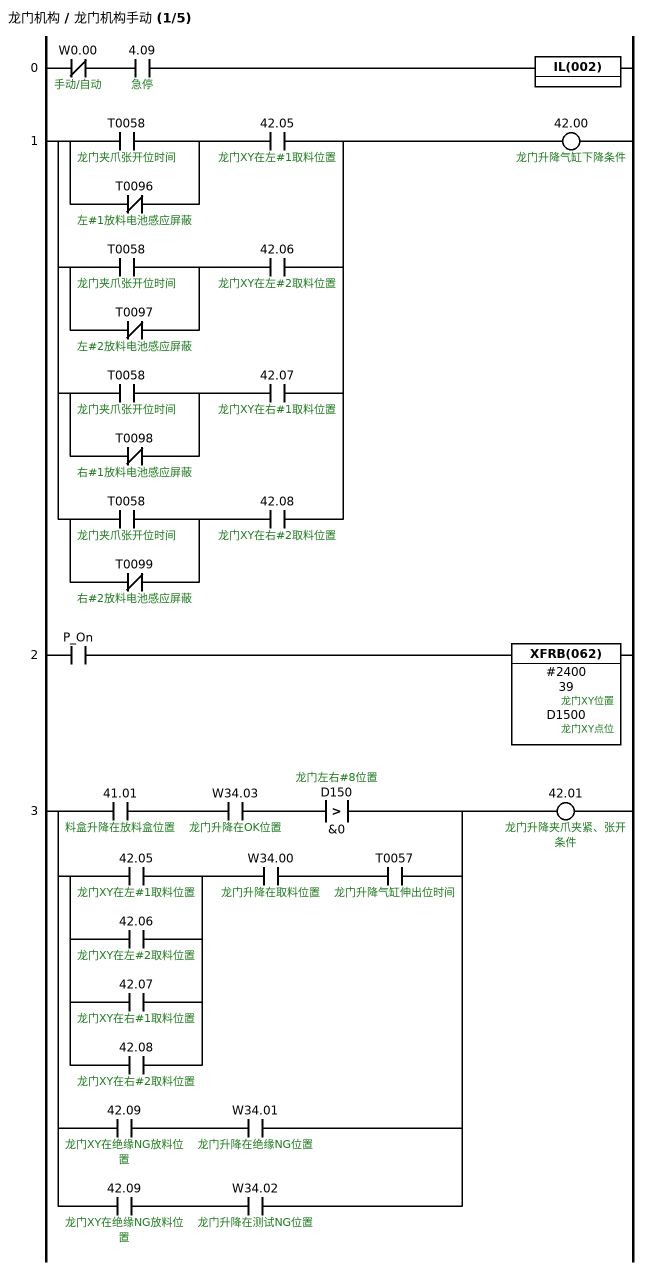
; rung 0
LDNOT W0.00  ; 手动/自动
AND 4.09  ; 急停
IL(002)
; rung 1
LD T0058  ; 龙门夹爪张开位时间
ORNOT T0096  ; 左#1放料电池感应屏蔽
AND 42.05  ; 龙门XY在左#1取料位置
LD T0058  ; 龙门夹爪张开位时间
ORNOT T0097  ; 左#2放料电池感应屏蔽
AND 42.06  ; 龙门XY在左#2取料位置
ORLD
LD T0058  ; 龙门夹爪张开位时间
ORNOT T0098  ; 右#1放料电池感应屏蔽
AND 42.07  ; 龙门XY在右#1取料位置
ORLD
LD T0058  ; 龙门夹爪张开位时间
ORNOT T0099  ; 右#2放料电池感应屏蔽
AND 42.08  ; 龙门XY在右#2取料位置
ORLD
OUT 42.00  ; 龙门升降气缸下降条件
; rung 2
LD P_On
XFRB(062) #2400 39 D1500  ; 龙门XY位置, 龙门XY点位
; rung 3
LD 41.01  ; 料盒升降在放料盒位置
AND W34.03  ; 龙门升降在OK位置
AND>L(321) D150 &0  ; 龙门左右#8位置
LD 42.05  ; 龙门XY在左#1取料位置
OR 42.06  ; 龙门XY在左#2取料位置
OR 42.07  ; 龙门XY在右#1取料位置
OR 42.08  ; 龙门XY在右#2取料位置
AND W34.00  ; 龙门升降在取料位置
AND T0057  ; 龙门升降气缸伸出位时间
ORLD
LD 42.09  ; 龙门XY在绝缘NG放料位置
AND W34.01  ; 龙门升降在绝缘NG位置
ORLD
LD 42.09  ; 龙门XY在绝缘NG放料位置
AND W34.02  ; 龙门升降在测试NG位置
ORLD
OUT 42.01  ; 龙门升降夹爪夹紧、张开条件

